{attribute 'GeneratedUsingTerminal: EK1100-0000-0018'}
{attribute addProperty BoxType "EK1100-0000-0018"}
{attribute addProperty Id "Beckhoff_EL31xxEK1122Beckhoff_EL31xxEK1122_183B25002A_0001_EL3101_0000_0016EL3101_123F62F814A_0002_EL3101_0000_0017EL3101_123F62F814A_0003_EL3101_0000_0018EL3101_123F62F814A_0004_EL3101_0000_0019EL3101_123F62F814A_0005_EL3102_0000_0000EL3102_5E13E83310A_0006_EL3102_0000_0016EL3102_FCC1BF8B24A_0007_EL3102_0000_0017EL3102_FCC1BF8B24A_0008_EL3102_0000_0018EL3102_FCC1BF8B24A_0009_EL3102_0000_0019EL3102_FCC1BF8B24A_0010_EL3102_0000_0020EL3102_FCC1BF8B24A_0011_EL3104_0000_0016EL3104_BE8A5C9E44A_0012_EL3104_0000_0017EL3104_BE8A5C9E44A_0013_EL3104_0000_0018EL3104_BE8A5C9E44A_0014_EL3104_0000_0019EL3104_BE8A5C9E44A_0015_EL3104_0000_0020EL3104_BE8A5C9E44A_0016_EL3111_0000_0016EL3111_123F62F814A_0017_EL3111_0000_0017EL3111_123F62F814A_0018_EL3111_0000_0018EL3111_123F62F814A_0019_EL3111_0000_0019EL3111_123F62F814A_0020_EL3111_0000_0020EL3111_123F62F814A_0021_EL3112_0000_0000EL3112_5E13E83310A_0022_EL3112_0000_0016EL3112_FCC1BF8B24A_0023_EL3112_0000_0017EL3112_FCC1BF8B24A_0024_EL3112_0000_0018EL3112_FCC1BF8B24A_0025_EL3112_0000_0019EL3112_FCC1BF8B24A_0026_EL3112_0011_0016EL3112_FCC1BF8B24A_0027_EL3114_0000_0016EL3114_BE8A5C9E44A_0028_EL3114_0000_0017EL3114_BE8A5C9E44A_0029_EL3114_0000_0018EL3114_BE8A5C9E44A_0030_EL3114_0000_0019EL3114_BE8A5C9E44A_0031_EL3114_0000_0020EL3114_BE8A5C9E44A_0032_EL3114_0000_0021EL3114_BE8A5C9E44A_0033_EL3121_0000_0016EL3121_123F62F814A_0034_EL3121_0000_0017EL3121_123F62F814A_0035_EL3121_0000_0018EL3121_123F62F814A_0036_EL3121_0000_0019EL3121_123F62F814A_0037_EL3122_0000_0000EL3122_5E13E83310A_0038_EL3122_0000_0016EL3122_FCC1BF8B24A_0039_EL3122_0000_0017EL3122_FCC1BF8B24A_0040_EL3122_0000_0018EL3122_FCC1BF8B24A_0041_EL3122_0000_0019EL3122_FCC1BF8B24A_0042_EL3124_0000_0016EL3124_BE8A5C9E44A_0043_EL3124_0000_0017EL3124_BE8A5C9E44A_0044_EL3124_0000_0018EL3124_BE8A5C9E44A_0045_EL3124_0000_0019EL3124_BE8A5C9E44A_0046_EL3124_0000_0020EL3124_BE8A5C9E44A_0047_EL3124_0090_0016EL3124_BE8A5C9E44A_0048_EL3141_0000_0016EL3141_123F62F814A_0049_EL3141_0000_0017EL3141_123F62F814A_0050_EL3141_0000_0018EL3141_123F62F814A_0051_EL3141_0000_0019EL3141_123F62F814A_0052_EL3141_0000_0020EL3141_123F62F814A_0053_EL3142_0000_0000EL3142_5E13E83310A_0054_EL3142_0000_0016EL3142_FCC1BF8B24A_0055_EL3142_0000_0017EL3142_FCC1BF8B24A_0056_EL3142_0000_0018EL3142_FCC1BF8B24A_0057_EL3142_0000_0019EL3142_FCC1BF8B24A_0058_EL3142_0010_0000EL3142_5E13E83310A_0059_EL3142_0010_0016EL3142_FCC1BF8B24A_0060_EL3142_0010_0017EL3142_FCC1BF8B24A_0061_EL3142_0010_0018EL3142_FCC1BF8B24A_0062_EL3142_0010_0019EL3142_FCC1BF8B24A_0063_EL3142_0010_0020EL3142_FCC1BF8B24A_0064_EL3142_0010_0021EL3142_FCC1BF8B24A_0065_EL3144_0000_0016EL3144_BE8A5C9E44A_0066_EL3144_0000_0017EL3144_BE8A5C9E44A_0067_EL3144_0000_0018EL3144_BE8A5C9E44A_0068_EL3144_0000_0019EL3144_BE8A5C9E44A_0069_EL3144_0000_0020EL3144_BE8A5C9E44A_0070_EL3151_0000_0016EL3151_123F62F814A_0071_EL3151_0000_0017EL3151_123F62F814A_0072_EL3151_0000_0018EL3151_123F62F814A_0073_EL3151_0000_0019EL3151_123F62F814A_0074_EL3151_0000_0020EL3151_123F62F814A_0075_EL3152_0000_0000EL3152_5E13E83310A_0076_EL3152_0000_0016EL3152_FCC1BF8B24A_0077_EL3152_0000_0017EL3152_FCC1BF8B24A_0078_EL3152_0000_0018EL3152_FCC1BF8B24A_0079_EL3152_0000_0019EL3152_FCC1BF8B24A_0080_EL3154_0000_0016EL3154_BE8A5C9E44A_0081_EL3154_0000_0017EL3154_BE8A5C9E44A_0082_EL3154_0000_0018EL3154_BE8A5C9E44A_0083_EL3154_0000_0019EL3154_BE8A5C9E44A_0084_EL3154_0000_0020EL3154_BE8A5C9E44A_0085_EL3161_0000_0016EL3161_123F62F814A_0086_EL3161_0000_0017EL3161_123F62F814A_0087_EL3161_0000_0018EL3161_123F62F814A_0088_EL3161_0000_0019EL3161_123F62F814A_0089_EL3162_0000_0000EL3162_5E13E83310A_0090_EL3162_0000_0016EL3162_FCC1BF8B24A_0091_EL3162_0000_0017EL3162_FCC1BF8B24A_0092_EL3162_0000_0018EL3162_FCC1BF8B24A_0093_EL3162_0000_0019EL3162_FCC1BF8B24A_0094_EL3164_0000_0016EL3164_BE8A5C9E44A_0095_EL3164_0000_0017EL3164_BE8A5C9E44A_0096_EL3164_0000_0018EL3164_BE8A5C9E44A_0097_EL3164_0000_0019EL3164_BE8A5C9E44A_0098_EL3164_0000_0020EL3164_BE8A5C9E44A_0099_EL3174_0000_0016EL3174_BE8A5C9E44A_0100_EL3174_0002_0017EL3174_BE8A5C9E44A_0101_EL3174_0032_0016EL3174_BE8A5C9E44A_0102_EL3174_0090_0016EL3174_BE8A5C9E44A_0103_EL3182_0000_0016EL3182_50349BB924A_0104_EL3182_0000_0017EL3182_50349BB924"}
{attribute addProperty CRC "2177961797"}
{attribute addProperty Size "2850"}
TYPE Beckhoff_EL31xx_81D10F45 EXTENDS EK1100_1FC0878B :
STRUCT
	{attribute addProperty Name "Beckhoff_EL31xxEK1122"}
	{attribute addProperty PreviousPort "Beckhoff EL31xx : B"}
	Beckhoff_EL31xxEK1122 : Beckhoff_EL31xxEK1122_183B2500;
	{attribute addProperty Name "A_0001_EL3101_0000_0016"}
	{attribute addProperty PreviousPort "Beckhoff EL31xxEK1122 : C"}
	A_0001_EL3101_0000_0016 : EL3101_123F62F8;
	{attribute addProperty Name "A_0002_EL3101_0000_0017"}
	{attribute addProperty PreviousPort "A_0001(EL3101-0000-0016) : B"}
	A_0002_EL3101_0000_0017 : EL3101_123F62F8;
	{attribute addProperty Name "A_0003_EL3101_0000_0018"}
	{attribute addProperty PreviousPort "A_0002(EL3101-0000-0017) : B"}
	A_0003_EL3101_0000_0018 : EL3101_123F62F8;
	{attribute addProperty Name "A_0004_EL3101_0000_0019"}
	{attribute addProperty PreviousPort "A_0003(EL3101-0000-0018) : B"}
	A_0004_EL3101_0000_0019 : EL3101_123F62F8;
	{attribute addProperty Name "A_0005_EL3102_0000_0000"}
	{attribute addProperty PreviousPort "A_0004(EL3101-0000-0019) : B"}
	A_0005_EL3102_0000_0000 : EL3102_5E13E833;
	{attribute addProperty Name "A_0006_EL3102_0000_0016"}
	{attribute addProperty PreviousPort "A_0005(EL3102-0000-0000) : B"}
	A_0006_EL3102_0000_0016 : EL3102_FCC1BF8B;
	{attribute addProperty Name "A_0007_EL3102_0000_0017"}
	{attribute addProperty PreviousPort "A_0006(EL3102-0000-0016) : B"}
	A_0007_EL3102_0000_0017 : EL3102_FCC1BF8B;
	{attribute addProperty Name "A_0008_EL3102_0000_0018"}
	{attribute addProperty PreviousPort "A_0007(EL3102-0000-0017) : B"}
	A_0008_EL3102_0000_0018 : EL3102_FCC1BF8B;
	{attribute addProperty Name "A_0009_EL3102_0000_0019"}
	{attribute addProperty PreviousPort "A_0008(EL3102-0000-0018) : B"}
	A_0009_EL3102_0000_0019 : EL3102_FCC1BF8B;
	{attribute addProperty Name "A_0010_EL3102_0000_0020"}
	{attribute addProperty PreviousPort "A_0009(EL3102-0000-0019) : B"}
	A_0010_EL3102_0000_0020 : EL3102_FCC1BF8B;
	{attribute addProperty Name "A_0011_EL3104_0000_0016"}
	{attribute addProperty PreviousPort "A_0010(EL3102-0000-0020) : B"}
	A_0011_EL3104_0000_0016 : EL3104_BE8A5C9E;
	{attribute addProperty Name "A_0012_EL3104_0000_0017"}
	{attribute addProperty PreviousPort "A_0011(EL3104-0000-0016) : B"}
	A_0012_EL3104_0000_0017 : EL3104_BE8A5C9E;
	{attribute addProperty Name "A_0013_EL3104_0000_0018"}
	{attribute addProperty PreviousPort "A_0012(EL3104-0000-0017) : B"}
	A_0013_EL3104_0000_0018 : EL3104_BE8A5C9E;
	{attribute addProperty Name "A_0014_EL3104_0000_0019"}
	{attribute addProperty PreviousPort "A_0013(EL3104-0000-0018) : B"}
	A_0014_EL3104_0000_0019 : EL3104_BE8A5C9E;
	{attribute addProperty Name "A_0015_EL3104_0000_0020"}
	{attribute addProperty PreviousPort "A_0014(EL3104-0000-0019) : B"}
	A_0015_EL3104_0000_0020 : EL3104_BE8A5C9E;
	{attribute addProperty Name "A_0016_EL3111_0000_0016"}
	{attribute addProperty PreviousPort "A_0015(EL3104-0000-0020) : B"}
	A_0016_EL3111_0000_0016 : EL3111_123F62F8;
	{attribute addProperty Name "A_0017_EL3111_0000_0017"}
	{attribute addProperty PreviousPort "A_0016(EL3111-0000-0016) : B"}
	A_0017_EL3111_0000_0017 : EL3111_123F62F8;
	{attribute addProperty Name "A_0018_EL3111_0000_0018"}
	{attribute addProperty PreviousPort "A_0017(EL3111-0000-0017) : B"}
	A_0018_EL3111_0000_0018 : EL3111_123F62F8;
	{attribute addProperty Name "A_0019_EL3111_0000_0019"}
	{attribute addProperty PreviousPort "A_0018(EL3111-0000-0018) : B"}
	A_0019_EL3111_0000_0019 : EL3111_123F62F8;
	{attribute addProperty Name "A_0020_EL3111_0000_0020"}
	{attribute addProperty PreviousPort "A_0019(EL3111-0000-0019) : B"}
	A_0020_EL3111_0000_0020 : EL3111_123F62F8;
	{attribute addProperty Name "A_0021_EL3112_0000_0000"}
	{attribute addProperty PreviousPort "A_0020(EL3111-0000-0020) : B"}
	A_0021_EL3112_0000_0000 : EL3112_5E13E833;
	{attribute addProperty Name "A_0022_EL3112_0000_0016"}
	{attribute addProperty PreviousPort "A_0021(EL3112-0000-0000) : B"}
	A_0022_EL3112_0000_0016 : EL3112_FCC1BF8B;
	{attribute addProperty Name "A_0023_EL3112_0000_0017"}
	{attribute addProperty PreviousPort "A_0022(EL3112-0000-0016) : B"}
	A_0023_EL3112_0000_0017 : EL3112_FCC1BF8B;
	{attribute addProperty Name "A_0024_EL3112_0000_0018"}
	{attribute addProperty PreviousPort "A_0023(EL3112-0000-0017) : B"}
	A_0024_EL3112_0000_0018 : EL3112_FCC1BF8B;
	{attribute addProperty Name "A_0025_EL3112_0000_0019"}
	{attribute addProperty PreviousPort "A_0024(EL3112-0000-0018) : B"}
	A_0025_EL3112_0000_0019 : EL3112_FCC1BF8B;
	{attribute addProperty Name "A_0026_EL3112_0011_0016"}
	{attribute addProperty PreviousPort "A_0025(EL3112-0000-0019) : B"}
	A_0026_EL3112_0011_0016 : EL3112_FCC1BF8B;
	{attribute addProperty Name "A_0027_EL3114_0000_0016"}
	{attribute addProperty PreviousPort "A_0026(EL3112-0011-0016) : B"}
	A_0027_EL3114_0000_0016 : EL3114_BE8A5C9E;
	{attribute addProperty Name "A_0028_EL3114_0000_0017"}
	{attribute addProperty PreviousPort "A_0027(EL3114-0000-0016) : B"}
	A_0028_EL3114_0000_0017 : EL3114_BE8A5C9E;
	{attribute addProperty Name "A_0029_EL3114_0000_0018"}
	{attribute addProperty PreviousPort "A_0028(EL3114-0000-0017) : B"}
	A_0029_EL3114_0000_0018 : EL3114_BE8A5C9E;
	{attribute addProperty Name "A_0030_EL3114_0000_0019"}
	{attribute addProperty PreviousPort "A_0029(EL3114-0000-0018) : B"}
	A_0030_EL3114_0000_0019 : EL3114_BE8A5C9E;
	{attribute addProperty Name "A_0031_EL3114_0000_0020"}
	{attribute addProperty PreviousPort "A_0030(EL3114-0000-0019) : B"}
	A_0031_EL3114_0000_0020 : EL3114_BE8A5C9E;
	{attribute addProperty Name "A_0032_EL3114_0000_0021"}
	{attribute addProperty PreviousPort "A_0031(EL3114-0000-0020) : B"}
	A_0032_EL3114_0000_0021 : EL3114_BE8A5C9E;
	{attribute addProperty Name "A_0033_EL3121_0000_0016"}
	{attribute addProperty PreviousPort "A_0032(EL3114-0000-0021) : B"}
	A_0033_EL3121_0000_0016 : EL3121_123F62F8;
	{attribute addProperty Name "A_0034_EL3121_0000_0017"}
	{attribute addProperty PreviousPort "A_0033(EL3121-0000-0016) : B"}
	A_0034_EL3121_0000_0017 : EL3121_123F62F8;
	{attribute addProperty Name "A_0035_EL3121_0000_0018"}
	{attribute addProperty PreviousPort "A_0034(EL3121-0000-0017) : B"}
	A_0035_EL3121_0000_0018 : EL3121_123F62F8;
	{attribute addProperty Name "A_0036_EL3121_0000_0019"}
	{attribute addProperty PreviousPort "A_0035(EL3121-0000-0018) : B"}
	A_0036_EL3121_0000_0019 : EL3121_123F62F8;
	{attribute addProperty Name "A_0037_EL3122_0000_0000"}
	{attribute addProperty PreviousPort "A_0036(EL3121-0000-0019) : B"}
	A_0037_EL3122_0000_0000 : EL3122_5E13E833;
	{attribute addProperty Name "A_0038_EL3122_0000_0016"}
	{attribute addProperty PreviousPort "A_0037(EL3122-0000-0000) : B"}
	A_0038_EL3122_0000_0016 : EL3122_FCC1BF8B;
	{attribute addProperty Name "A_0039_EL3122_0000_0017"}
	{attribute addProperty PreviousPort "A_0038(EL3122-0000-0016) : B"}
	A_0039_EL3122_0000_0017 : EL3122_FCC1BF8B;
	{attribute addProperty Name "A_0040_EL3122_0000_0018"}
	{attribute addProperty PreviousPort "A_0039(EL3122-0000-0017) : B"}
	A_0040_EL3122_0000_0018 : EL3122_FCC1BF8B;
	{attribute addProperty Name "A_0041_EL3122_0000_0019"}
	{attribute addProperty PreviousPort "A_0040(EL3122-0000-0018) : B"}
	A_0041_EL3122_0000_0019 : EL3122_FCC1BF8B;
	{attribute addProperty Name "A_0042_EL3124_0000_0016"}
	{attribute addProperty PreviousPort "A_0041(EL3122-0000-0019) : B"}
	A_0042_EL3124_0000_0016 : EL3124_BE8A5C9E;
	{attribute addProperty Name "A_0043_EL3124_0000_0017"}
	{attribute addProperty PreviousPort "A_0042(EL3124-0000-0016) : B"}
	A_0043_EL3124_0000_0017 : EL3124_BE8A5C9E;
	{attribute addProperty Name "A_0044_EL3124_0000_0018"}
	{attribute addProperty PreviousPort "A_0043(EL3124-0000-0017) : B"}
	A_0044_EL3124_0000_0018 : EL3124_BE8A5C9E;
	{attribute addProperty Name "A_0045_EL3124_0000_0019"}
	{attribute addProperty PreviousPort "A_0044(EL3124-0000-0018) : B"}
	A_0045_EL3124_0000_0019 : EL3124_BE8A5C9E;
	{attribute addProperty Name "A_0046_EL3124_0000_0020"}
	{attribute addProperty PreviousPort "A_0045(EL3124-0000-0019) : B"}
	A_0046_EL3124_0000_0020 : EL3124_BE8A5C9E;
	{attribute addProperty Name "A_0047_EL3124_0090_0016"}
	{attribute addProperty PreviousPort "A_0046(EL3124-0000-0020) : B"}
	A_0047_EL3124_0090_0016 : EL3124_BE8A5C9E;
	{attribute addProperty Name "A_0048_EL3141_0000_0016"}
	{attribute addProperty PreviousPort "A_0047(EL3124-0090-0016) : B"}
	A_0048_EL3141_0000_0016 : EL3141_123F62F8;
	{attribute addProperty Name "A_0049_EL3141_0000_0017"}
	{attribute addProperty PreviousPort "A_0048(EL3141-0000-0016) : B"}
	A_0049_EL3141_0000_0017 : EL3141_123F62F8;
	{attribute addProperty Name "A_0050_EL3141_0000_0018"}
	{attribute addProperty PreviousPort "A_0049(EL3141-0000-0017) : B"}
	A_0050_EL3141_0000_0018 : EL3141_123F62F8;
	{attribute addProperty Name "A_0051_EL3141_0000_0019"}
	{attribute addProperty PreviousPort "A_0050(EL3141-0000-0018) : B"}
	A_0051_EL3141_0000_0019 : EL3141_123F62F8;
	{attribute addProperty Name "A_0052_EL3141_0000_0020"}
	{attribute addProperty PreviousPort "A_0051(EL3141-0000-0019) : B"}
	A_0052_EL3141_0000_0020 : EL3141_123F62F8;
	{attribute addProperty Name "A_0053_EL3142_0000_0000"}
	{attribute addProperty PreviousPort "A_0052(EL3141-0000-0020) : B"}
	A_0053_EL3142_0000_0000 : EL3142_5E13E833;
	{attribute addProperty Name "A_0054_EL3142_0000_0016"}
	{attribute addProperty PreviousPort "A_0053(EL3142-0000-0000) : B"}
	A_0054_EL3142_0000_0016 : EL3142_FCC1BF8B;
	{attribute addProperty Name "A_0055_EL3142_0000_0017"}
	{attribute addProperty PreviousPort "A_0054(EL3142-0000-0016) : B"}
	A_0055_EL3142_0000_0017 : EL3142_FCC1BF8B;
	{attribute addProperty Name "A_0056_EL3142_0000_0018"}
	{attribute addProperty PreviousPort "A_0055(EL3142-0000-0017) : B"}
	A_0056_EL3142_0000_0018 : EL3142_FCC1BF8B;
	{attribute addProperty Name "A_0057_EL3142_0000_0019"}
	{attribute addProperty PreviousPort "A_0056(EL3142-0000-0018) : B"}
	A_0057_EL3142_0000_0019 : EL3142_FCC1BF8B;
	{attribute addProperty Name "A_0058_EL3142_0010_0000"}
	{attribute addProperty PreviousPort "A_0057(EL3142-0000-0019) : B"}
	A_0058_EL3142_0010_0000 : EL3142_5E13E833;
	{attribute addProperty Name "A_0059_EL3142_0010_0016"}
	{attribute addProperty PreviousPort "A_0058(EL3142-0010-0000) : B"}
	A_0059_EL3142_0010_0016 : EL3142_FCC1BF8B;
	{attribute addProperty Name "A_0060_EL3142_0010_0017"}
	{attribute addProperty PreviousPort "A_0059(EL3142-0010-0016) : B"}
	A_0060_EL3142_0010_0017 : EL3142_FCC1BF8B;
	{attribute addProperty Name "A_0061_EL3142_0010_0018"}
	{attribute addProperty PreviousPort "A_0060(EL3142-0010-0017) : B"}
	A_0061_EL3142_0010_0018 : EL3142_FCC1BF8B;
	{attribute addProperty Name "A_0062_EL3142_0010_0019"}
	{attribute addProperty PreviousPort "A_0061(EL3142-0010-0018) : B"}
	A_0062_EL3142_0010_0019 : EL3142_FCC1BF8B;
	{attribute addProperty Name "A_0063_EL3142_0010_0020"}
	{attribute addProperty PreviousPort "A_0062(EL3142-0010-0019) : B"}
	A_0063_EL3142_0010_0020 : EL3142_FCC1BF8B;
	{attribute addProperty Name "A_0064_EL3142_0010_0021"}
	{attribute addProperty PreviousPort "A_0063(EL3142-0010-0020) : B"}
	A_0064_EL3142_0010_0021 : EL3142_FCC1BF8B;
	{attribute addProperty Name "A_0065_EL3144_0000_0016"}
	{attribute addProperty PreviousPort "A_0064(EL3142-0010-0021) : B"}
	A_0065_EL3144_0000_0016 : EL3144_BE8A5C9E;
	{attribute addProperty Name "A_0066_EL3144_0000_0017"}
	{attribute addProperty PreviousPort "A_0065(EL3144-0000-0016) : B"}
	A_0066_EL3144_0000_0017 : EL3144_BE8A5C9E;
	{attribute addProperty Name "A_0067_EL3144_0000_0018"}
	{attribute addProperty PreviousPort "A_0066(EL3144-0000-0017) : B"}
	A_0067_EL3144_0000_0018 : EL3144_BE8A5C9E;
	{attribute addProperty Name "A_0068_EL3144_0000_0019"}
	{attribute addProperty PreviousPort "A_0067(EL3144-0000-0018) : B"}
	A_0068_EL3144_0000_0019 : EL3144_BE8A5C9E;
	{attribute addProperty Name "A_0069_EL3144_0000_0020"}
	{attribute addProperty PreviousPort "A_0068(EL3144-0000-0019) : B"}
	A_0069_EL3144_0000_0020 : EL3144_BE8A5C9E;
	{attribute addProperty Name "A_0070_EL3151_0000_0016"}
	{attribute addProperty PreviousPort "A_0069(EL3144-0000-0020) : B"}
	A_0070_EL3151_0000_0016 : EL3151_123F62F8;
	{attribute addProperty Name "A_0071_EL3151_0000_0017"}
	{attribute addProperty PreviousPort "A_0070(EL3151-0000-0016) : B"}
	A_0071_EL3151_0000_0017 : EL3151_123F62F8;
	{attribute addProperty Name "A_0072_EL3151_0000_0018"}
	{attribute addProperty PreviousPort "A_0071(EL3151-0000-0017) : B"}
	A_0072_EL3151_0000_0018 : EL3151_123F62F8;
	{attribute addProperty Name "A_0073_EL3151_0000_0019"}
	{attribute addProperty PreviousPort "A_0072(EL3151-0000-0018) : B"}
	A_0073_EL3151_0000_0019 : EL3151_123F62F8;
	{attribute addProperty Name "A_0074_EL3151_0000_0020"}
	{attribute addProperty PreviousPort "A_0073(EL3151-0000-0019) : B"}
	A_0074_EL3151_0000_0020 : EL3151_123F62F8;
	{attribute addProperty Name "A_0075_EL3152_0000_0000"}
	{attribute addProperty PreviousPort "A_0074(EL3151-0000-0020) : B"}
	A_0075_EL3152_0000_0000 : EL3152_5E13E833;
	{attribute addProperty Name "A_0076_EL3152_0000_0016"}
	{attribute addProperty PreviousPort "A_0075(EL3152-0000-0000) : B"}
	A_0076_EL3152_0000_0016 : EL3152_FCC1BF8B;
	{attribute addProperty Name "A_0077_EL3152_0000_0017"}
	{attribute addProperty PreviousPort "A_0076(EL3152-0000-0016) : B"}
	A_0077_EL3152_0000_0017 : EL3152_FCC1BF8B;
	{attribute addProperty Name "A_0078_EL3152_0000_0018"}
	{attribute addProperty PreviousPort "A_0077(EL3152-0000-0017) : B"}
	A_0078_EL3152_0000_0018 : EL3152_FCC1BF8B;
	{attribute addProperty Name "A_0079_EL3152_0000_0019"}
	{attribute addProperty PreviousPort "A_0078(EL3152-0000-0018) : B"}
	A_0079_EL3152_0000_0019 : EL3152_FCC1BF8B;
	{attribute addProperty Name "A_0080_EL3154_0000_0016"}
	{attribute addProperty PreviousPort "A_0079(EL3152-0000-0019) : B"}
	A_0080_EL3154_0000_0016 : EL3154_BE8A5C9E;
	{attribute addProperty Name "A_0081_EL3154_0000_0017"}
	{attribute addProperty PreviousPort "A_0080(EL3154-0000-0016) : B"}
	A_0081_EL3154_0000_0017 : EL3154_BE8A5C9E;
	{attribute addProperty Name "A_0082_EL3154_0000_0018"}
	{attribute addProperty PreviousPort "A_0081(EL3154-0000-0017) : B"}
	A_0082_EL3154_0000_0018 : EL3154_BE8A5C9E;
	{attribute addProperty Name "A_0083_EL3154_0000_0019"}
	{attribute addProperty PreviousPort "A_0082(EL3154-0000-0018) : B"}
	A_0083_EL3154_0000_0019 : EL3154_BE8A5C9E;
	{attribute addProperty Name "A_0084_EL3154_0000_0020"}
	{attribute addProperty PreviousPort "A_0083(EL3154-0000-0019) : B"}
	A_0084_EL3154_0000_0020 : EL3154_BE8A5C9E;
	{attribute addProperty Name "A_0085_EL3161_0000_0016"}
	{attribute addProperty PreviousPort "A_0084(EL3154-0000-0020) : B"}
	A_0085_EL3161_0000_0016 : EL3161_123F62F8;
	{attribute addProperty Name "A_0086_EL3161_0000_0017"}
	{attribute addProperty PreviousPort "A_0085(EL3161-0000-0016) : B"}
	A_0086_EL3161_0000_0017 : EL3161_123F62F8;
	{attribute addProperty Name "A_0087_EL3161_0000_0018"}
	{attribute addProperty PreviousPort "A_0086(EL3161-0000-0017) : B"}
	A_0087_EL3161_0000_0018 : EL3161_123F62F8;
	{attribute addProperty Name "A_0088_EL3161_0000_0019"}
	{attribute addProperty PreviousPort "A_0087(EL3161-0000-0018) : B"}
	A_0088_EL3161_0000_0019 : EL3161_123F62F8;
	{attribute addProperty Name "A_0089_EL3162_0000_0000"}
	{attribute addProperty PreviousPort "A_0088(EL3161-0000-0019) : B"}
	A_0089_EL3162_0000_0000 : EL3162_5E13E833;
	{attribute addProperty Name "A_0090_EL3162_0000_0016"}
	{attribute addProperty PreviousPort "A_0089(EL3162-0000-0000) : B"}
	A_0090_EL3162_0000_0016 : EL3162_FCC1BF8B;
	{attribute addProperty Name "A_0091_EL3162_0000_0017"}
	{attribute addProperty PreviousPort "A_0090(EL3162-0000-0016) : B"}
	A_0091_EL3162_0000_0017 : EL3162_FCC1BF8B;
	{attribute addProperty Name "A_0092_EL3162_0000_0018"}
	{attribute addProperty PreviousPort "A_0091(EL3162-0000-0017) : B"}
	A_0092_EL3162_0000_0018 : EL3162_FCC1BF8B;
	{attribute addProperty Name "A_0093_EL3162_0000_0019"}
	{attribute addProperty PreviousPort "A_0092(EL3162-0000-0018) : B"}
	A_0093_EL3162_0000_0019 : EL3162_FCC1BF8B;
	{attribute addProperty Name "A_0094_EL3164_0000_0016"}
	{attribute addProperty PreviousPort "A_0093(EL3162-0000-0019) : B"}
	A_0094_EL3164_0000_0016 : EL3164_BE8A5C9E;
	{attribute addProperty Name "A_0095_EL3164_0000_0017"}
	{attribute addProperty PreviousPort "A_0094(EL3164-0000-0016) : B"}
	A_0095_EL3164_0000_0017 : EL3164_BE8A5C9E;
	{attribute addProperty Name "A_0096_EL3164_0000_0018"}
	{attribute addProperty PreviousPort "A_0095(EL3164-0000-0017) : B"}
	A_0096_EL3164_0000_0018 : EL3164_BE8A5C9E;
	{attribute addProperty Name "A_0097_EL3164_0000_0019"}
	{attribute addProperty PreviousPort "A_0096(EL3164-0000-0018) : B"}
	A_0097_EL3164_0000_0019 : EL3164_BE8A5C9E;
	{attribute addProperty Name "A_0098_EL3164_0000_0020"}
	{attribute addProperty PreviousPort "A_0097(EL3164-0000-0019) : B"}
	A_0098_EL3164_0000_0020 : EL3164_BE8A5C9E;
	{attribute addProperty Name "A_0099_EL3174_0000_0016"}
	{attribute addProperty PreviousPort "A_0098(EL3164-0000-0020) : B"}
	A_0099_EL3174_0000_0016 : EL3174_BE8A5C9E;
	{attribute addProperty Name "A_0100_EL3174_0002_0017"}
	{attribute addProperty PreviousPort "A_0099(EL3174-0000-0016) : B"}
	A_0100_EL3174_0002_0017 : EL3174_BE8A5C9E;
	{attribute addProperty Name "A_0101_EL3174_0032_0016"}
	{attribute addProperty PreviousPort "A_0100(EL3174-0002-0017) : B"}
	A_0101_EL3174_0032_0016 : EL3174_BE8A5C9E;
	{attribute addProperty Name "A_0102_EL3174_0090_0016"}
	{attribute addProperty PreviousPort "A_0101(EL3174-0032-0016) : B"}
	A_0102_EL3174_0090_0016 : EL3174_BE8A5C9E;
	{attribute addProperty Name "A_0103_EL3182_0000_0016"}
	{attribute addProperty PreviousPort "A_0102(EL3174-0090-0016) : B"}
	A_0103_EL3182_0000_0016 : EL3182_50349BB9;
	{attribute addProperty Name "A_0104_EL3182_0000_0017"}
	{attribute addProperty PreviousPort "A_0103(EL3182-0000-0016) : B"}
	A_0104_EL3182_0000_0017 : EL3182_50349BB9;
END_STRUCT
END_TYPE

(* stored: Version 1.2.0.0, ProductVersion 3.1.4024.9
   DUT Beckhoff_EL31xx_81D10F45: Id {afec1317-2a33-40c3-878f-88cef5ffe423} *)
